// TIA Portal V17 export
// export: Created 2024-08-20T13:26:10.6182293Z, ExportSetting WithDefaults, DisplayName Totally Integrated Automation Portal, DisplayVersion V17 Update 4, DisplayName TIA Portal Openness, DisplayVersion V17 Update 4, DisplayName TIA Portal Version Control Interface, DisplayVersion V17, DisplayName STEP 7 Professional, DisplayVersion V17 Update 4, DisplayName STEP 7 Safety, DisplayVersion V17, DisplayName WinCC Advanced, DisplayVersion V17 Update 4
DATA_BLOCK "SETPOINTS"   // DB305
{ S7_Optimized_Access := 'FALSE' }
VERSION : 0.1
// stored: AutoNumber false, DBAccessibleFromOPCUA true, IsOnlyStoredInLoadMemory false, IsWriteProtectedInAS false
   VAR RETAIN
      "MB-01-SP" : Real := 60.0;   // Setpoint manual elevatoria principal
      "MB-02-SP" : Real := 0.0;   // Setpoint manual elevatoria principal
      "MB-03-SP" : Real := 60.0;   // Setpoint manual elevatoria principal
      "MB-04-SP" : Real := 60.0;   // Setpoint manual elevatoria principal
      "LIT_001-SPHH" : Real := 90.0;   // Setpoint muito alto elevatoria principal
      "LIT_001-SPH" : Real := 70.0;   // Setpoint nível alto elevatoria principal
      "LIT_001-SPL" : Real := 10.0;   // Setpoint nível baixo elevatoria principal
      "LIT_001-SPLL" : Real := 0.0;   // Setpoint nível muito baixo elevatoria principal
      "LIT_001-SPM" : Real := 48.0;   // Habilita valor manual para medidor
      "LIT_001-SPC" : Real := 0.0;   // Setpoint de controle tanque
      "LIT-001-P" : Real := 0.0;
      SP_NVL_MIN : Real := 1.0;   // setpoint nivel minimo do tanque para proteção hidraulica
      "MB-P-SP-DL" : Real := 2.0;   // Setpoint para desligar bomba Principal
      "MB-P-SP-L" : Real := 2.6;   // Setpoint para ligar bomba Principal
      "MB-C1-SP-DL" : Real := 2.35;   // Setpoint para desligar bomba complementar 1
      "MB-C1-SP-L" : Real := 2.9;   // Setpoint para ligar bomba complementar 1
      "MB-C2-SP-DL" : Real := 2.66;   // Setpoint para desligar bomba complementar 2
      "MB-C2-SP-L" : Real := 3.9;   // Setpoint para ligar bomba complementar 2
      "MB-C3-SP-DL" : Real := 0.0;   // Setpoint para desligar bomba complementar 3
      "MB-C3-SP-L" : Real := 0.0;   // Setpoint para ligar bomba complementar 3
   END_VAR
BEGIN
END_DATA_BLOCK
